Yaskawa INFORM job: TESR2.JBI

/JOB
//NAME TESR2
//POS
///NPOS 1,1,0,0,0,0
///TOOL 0
///POSTYPE PULSE
///PULSE
C00000=-6929,-138827,-107581,-17031,60703,17870
BC00000=161140,743111,242028
//INST
///DATE 2024/01/25 09:48
///ATTR SC,RW
///GROUP1 RB1,BS1
NOP
MOVJ C00000 BC00000 VJ=0.78
END
